PROGRAM V0_7
VAR
	bOn : BOOL;
	bOff : BOOL;
END_VAR
(*
	Teleruptorschakeling | uitleg
	
	In woningen wordt een soortgelijke schakeling gebruikt om de verlichting in en uit te schakelen door gebruik te maken van parallel geschakelde drukknoppen. Men noemt het ook soms een afstands- of trappenhuisschakelaar. Maak deze na in LADDER en probeer te achterhalen hoe deze werkt.

	Zorg ervoor dat er meerdere drukknoppen (op ieder verdiep) gebruikt kunnen worden.

	De P in het maakcontact Ingang zorgt ervoor dat deze puls- of flank-gestuurd is. Deze kan je eenvoudig toevoegen door het maakcontact te selecteren en de P-toets op je toetsenbord in te drukken.

	De tussenvariable M0 wordt in de PLC wereld een Merker genoemd. Deze is nodig omdat je in LADDER een maakcontact niet kan inverteren alsook flankgestuurd maken.

	Je zal wel gemerkt hebben dat in het tweede netwerk de NO maakcontact lamp parallel met NO maakcontact M0 als een overneemcontact werkt. De NC merker M0 en NC lamp die omgekeerd in serie staan zorgen ervoor dat dit onderbroken kan worden
*)
VAR // added by the converter: edge detectors and wires of the graphical bodies
    _rt1, _rt2, _rt3, _rt4 : R_TRIG;
END_VAR

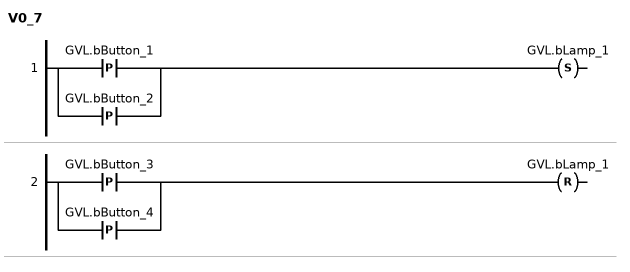
// NETWORK 1
_rt1(CLK := GVL.bButton_1);
_rt2(CLK := GVL.bButton_2);
GVL.bLamp_1 S= _rt1.Q OR _rt2.Q;

// NETWORK 2
_rt3(CLK := GVL.bButton_3);
_rt4(CLK := GVL.bButton_4);
GVL.bLamp_1 R= _rt3.Q OR _rt4.Q;

END_PROGRAM

(* stored: Version 1.1.0.1, ProductVersion 3.1.4024.12
   POU V0_7: Id {1317fce5-6d05-4a7d-a34e-8d1e185c12e9}, SpecialFunc None *)
